// TwinCAT 3 PLC project _10_Adapter
// ProgramVersion: 3.1.4023.0
// libraries:
//   Tc2_Standard, * (Beckhoff Automation GmbH)
//   Tc2_System, * (Beckhoff Automation GmbH)
//   Tc3_Module, * (Beckhoff Automation GmbH)
// project tree:
//   Adapter Pattern/Adapter/ CylinderVtem.TcPOU
//   Adapter Pattern/Festo/ IVtemByFesto.TcIO, VtemByFesto.TcPOU
//   Adapter Pattern/ P_Adapter.TcPOU
//   Adapter Pattern/Standard/ Cylinder.TcPOU, ICylinder.TcIO
//   / MAIN.TcPOU, PlcTask.TcTTO
// (motion and I/O tree: see PLC project 13_decorator)
// real-time tasks:
//   TASK PlcTask: cycle T#10ms, priority 20, ADS port 350
// variable links:

CONFIGURATION _10_Adapter
    RESOURCE PLC ON TwinCAT3
        TASK PlcTask(INTERVAL := T#10ms, PRIORITY := 20);
        PROGRAM MAIN WITH PlcTask : MAIN;
    END_RESOURCE
END_CONFIGURATION

// ---- Adapter Pattern/Festo/IVtemByFesto.TcIO
INTERFACE IVtemByFesto

METHOD moveBwd : BOOL
VAR_INPUT
END_VAR
END_METHOD

METHOD moveFwd : BOOL
VAR_INPUT
END_VAR
END_METHOD

END_INTERFACE

// ---- Adapter Pattern/Standard/ICylinder.TcIO
INTERFACE ICylinder

METHOD bwd
VAR_INPUT
END_VAR
END_METHOD

METHOD fwd
VAR_INPUT
END_VAR
END_METHOD

END_INTERFACE

// ---- MAIN.TcPOU
PROGRAM MAIN
VAR
END_VAR

(* 
	GOF 		Convert the interface of a class into another interface clients expect. Adapter
				lets classes work together that couldn't otherwise because of incompatible
				interfaces.
*)
P_Adapter();

END_PROGRAM

// ---- Adapter Pattern/P_Adapter.TcPOU
PROGRAM P_Adapter
VAR
	cylinderStandard				: Cylinder;
	cylinderVtem					: CylinderVtem;
END_VAR


// Move cylinders forward
cylinderStandard.fwd();
cylinderVtem.fwd();

END_PROGRAM

// ---- Adapter Pattern/Standard/Cylinder.TcPOU
FUNCTION_BLOCK Cylinder IMPLEMENTS ICylinder
VAR_INPUT
END_VAR
VAR_OUTPUT
END_VAR
VAR
END_VAR

{warning 'add method implementation '}
METHOD bwd
END_METHOD

{warning 'add method implementation '}
METHOD fwd
END_METHOD

END_FUNCTION_BLOCK

// ---- Adapter Pattern/Adapter/CylinderVtem.TcPOU
FUNCTION_BLOCK CylinderVtem IMPLEMENTS ICylinder
VAR
	vtem				: VtemByFesto;
END_VAR

;

METHOD bwd
vtem.moveBwd();
END_METHOD

METHOD fwd
vtem.moveFwd();
END_METHOD

END_FUNCTION_BLOCK

// ---- Adapter Pattern/Festo/VtemByFesto.TcPOU
FUNCTION_BLOCK VtemByFesto IMPLEMENTS IVtemByFesto
VAR_INPUT
END_VAR
VAR_OUTPUT
END_VAR
VAR
END_VAR

{warning 'add method implementation '}
METHOD moveBwd : BOOL
END_METHOD

{warning 'add method implementation '}
METHOD moveFwd : BOOL
END_METHOD

END_FUNCTION_BLOCK
